    //========================Manual=============================
    modesMachine         := eMachineModes.Manual;
    expectedColor.Green  := FALSE;
    expectedColor.Red    := FALSE;
    expectedColor.Yellow := TRUE;

    actualColor := itfDut.SetMachineMode(modesMachine);

    AssertEquals
    (
        Expected  := expectedColor
        , Actual  := actualColor
        , Message := 'ColorOuput shall be Yellow'
    );

    //========================Fault=============================
    modesMachine         := eMachineModes.Fault;
    expectedColor.Green  := FALSE;
    expectedColor.Red    := TRUE;
    expectedColor.Yellow := FALSE;

     itfDut.SetMachineMode(modesMachine);
     actualColor := itfDut.GetColorsSignalLightMachineModes;
    AssertEquals
    (
        Expected  := expectedColor
        , Actual  := actualColor
        , Message := 'ColorOuput shall be Red'
    );

    state := 10;
END_IF

IF state = 10 THEN

    //========================Home=============================
    modesMachine := eMachineModes.Home;
    itfDut.SetMachineMode(modesMachine);

    IF eMachineModes.Home = modesMachine THEN
        timer(in := TRUE);
    END_IF

    expectedColor.Red    := FALSE;
    expectedColor.Yellow := FALSE;

    IF timer.ET >= 0 * blinkTime AND timer.ET < blinkTime THEN
        expectedColor.Green := TRUE;
        actualColor         := itfDut.SetMachineMode(modesMachine);

        AssertEquals
        (
            Expected  := expectedColor
            , Actual  := actualColor
            , Message := 'ColorOuput shall be GreenBlinking and True 1 '
        );

    ELSIF timer.ET > blinkTime + T#2MS AND timer.ET < 2 * blinkTime THEN
        expectedColor.Green := FALSE;
        actualColor         := itfDut.SetMachineMode(modesMachine);

        AssertEquals
        (
            Expected  := expectedColor
            , Actual  := actualColor
            , Message := 'ColorOuput shall be GreenBlinking and False 2'
        );

    ELSIF timer.ET > 2 * blinkTime + T#2MS AND timer.ET < 3 * blinkTime THEN
        expectedColor.Green := TRUE;
        actualColor         := itfDut.SetMachineMode(modesMachine);

        AssertEquals
        (
            Expected  := expectedColor
            , Actual  := actualColor
            , Message := 'ColorOuput shall be GreenBlinking and TRUE 3'
        );
    ELSIF timer.ET > 3 * blinkTime + T#2MS AND timer.ET < 4 * blinkTime THEN
        expectedColor.Green := False;
        actualColor         := itfDut.SetMachineMode(modesMachine);

        AssertEquals
        (
            Expected  := expectedColor
            , Actual  := actualColor
            , Message := 'ColorOuput shall be GreenBlinking and TRUE 4'
        );
    ELSIF timer.ET > 5 * blinkTime THEN

        //========================Idle, Check again if all out =============================
        modesMachine := eMachineModes.Idle;

        expectedColor.Green  := FALSE;
        expectedColor.Red    := FALSE;
        expectedColor.Yellow := FALSE;

        actualColor := itfDut.SetMachineMode(modesMachine);

        AssertEquals
        (
            Expected  := expectedColor
            , Actual  := actualColor
            , Message := 'ColorOuput shall be Off again'
        );

        {analysis -9}
        TEST_FINISHED();
    END_IF
END_IF
END_METHOD

PROPERTY StartCycleCount : ULINT
GET
StartCycleCount := THIS^._nfContext._startCycleCount;
END_GET
END_PROPERTY

END_FUNCTION_BLOCK

// ---- POUs/SignalLights MachineStatus/POUs/SignalLightsController.TcPOU
FUNCTION_BLOCK SignalLightsController EXTENDS TcoCore.TcoObject IMPLEMENTS ISignalLightsController
VAR
    blinker : Blinker;
    colorsStatus : ColorsSignalLightsStatus;
    colorsMode : ColorsSignalLightMachineModes;
END_VAR

METHOD FB_init : BOOL
VAR_INPUT
    bInitRetains : BOOL; // if TRUE, the retain variables are initialized (warm start / cold start)
    bInCopyCode  : BOOL; // if TRUE, the instance afterwards gets moved into the copy code (online change)
    ParentObject : ITcoObject;
END_VAR
END_METHOD

PROPERTY GetColorsSignalLightMachineModes :  ColorsSignalLightMachineModes
GET
GetColorsSignalLightMachineModes := colorsMode;
END_GET
END_PROPERTY

PROPERTY GetColorsSignalLightMachineStatus : ColorsSignalLightsStatus
GET
GetColorsSignalLightMachineStatus := colorsStatus;
END_GET
END_PROPERTY

(*~
    <docu>
        <summary>
            Restore all tasks of this instance into initial state.
        </summary>
    </docu>
~*)
METHOD Restore : ITcoRestorable
END_METHOD

METHOD PROTECTED ServiceMode
END_METHOD

METHOD SetBlinkTime
VAR_INPUT
    blinkOnTime  : TIME;
    blinkOffTime : TIME;
END_VAR
THIS^.blinker.SetOffTime(blinkOffTime);
THIS^.blinker.SetOnTime(blinkOnTime);
END_METHOD

METHOD SetMachineMode : ColorsSignalLightMachineModes
VAR_INPUT
    currentMachineMode : eMachineModes ;
END_VAR

IF eMachineModes.Home = currentMachineMode THEN
    blinker.ExecuteTimer();
END_IF

CASE currentMachineMode OF
    eMachineModes.Fault:
        colorsMode.Red    := TRUE;
        colorsMode.Green  := FALSE;
        colorsMode.Yellow := FALSE;

    eMachineModes.Idle:

        colorsMode.Red    := FALSE;
        colorsMode.Green  := FALSE;
        colorsMode.Yellow := FALSE;

    eMachineModes.Automat:
        colorsMode.Red    := FALSE;
        colorsMode.Green  := TRUE;
        colorsMode.Yellow := FALSE;

    eMachineModes.Step:
        colorsMode.Red    := FALSE;
        colorsMode.Green  := TRUE;
        colorsMode.Yellow := TRUE;

    eMachineModes.Home:
        colorsMode.Red    := FALSE;
        colorsMode.Yellow := FALSE;
        colorsMode.Green  := blinker.IsOn;

    eMachineModes.Manual:
        colorsMode.Red    := FALSE;
        colorsMode.Yellow := TRUE;
        colorsMode.Green  := FALSE;
ELSE
    ;
END_CASE

 SetMachineMode := colorsMode ;
END_METHOD

METHOD SetMachineStatusOff : ColorsSignalLightsStatus
VAR_INPUT
    currentMachineStatus : eMachineStatus;
END_VAR
CASE currentMachineStatus OF
    eMachineStatus.Blue:
        colorsStatus.Blue := FALSE;
    eMachineStatus.Turquise:
        colorsStatus.Turquise := FALSE;
    eMachineStatus.Violet:
        colorsStatus.Violet := FALSE;
    eMachineStatus.White:
        colorsStatus.White := FALSE;
    eMachineStatus.All:
        colorsStatus.Blue     := FALSE;
        colorsStatus.Turquise := FALSE;
        colorsStatus.White    := FALSE;
        colorsStatus.Violet   := FALSE;
END_CASE

SetMachineStatusOff := colorsStatus;
END_METHOD

METHOD SetMachineStatusOn : ColorsSignalLightsStatus
VAR_INPUT
    currentMachineStatus : eMachineStatus;
END_VAR
CASE currentMachineStatus OF
    eMachineStatus.Blue:
        colorsStatus.Blue := TRUE;
    eMachineStatus.Turquise:
        colorsStatus.Turquise := TRUE;
    eMachineStatus.Violet:
        colorsStatus.Violet := TRUE;
    eMachineStatus.White:
        colorsStatus.White := TRUE;
    eMachineStatus.All:
        colorsStatus.Blue     := TRUE;
        colorsStatus.Turquise := TRUE;
        colorsStatus.White    := TRUE;
        colorsStatus.Violet   := TRUE;
END_CASE

SetMachineStatusOn := colorsStatus;
END_METHOD

END_FUNCTION_BLOCK

// ---- POUs/Utilities/Blinker.TcPOU
FUNCTION_BLOCK Blinker
VAR
    _offTime : TIME := T#1000MS;
    _onTime  : TIME := T#1000MS;
    onTimer : TON;
    offTimer : TON;
    blinkOutput : BOOL;
    state : INT ;
END_VAR

METHOD ExecuteTimer : BOOL
VAR_INPUT
END_VAR
IF state = 0 THEN
    onTimer(in := FALSE);
    offTimer(in := FALSE);

    state := 10;
END_IF

IF state = 10 THEN
    onTimer(in := TRUE, pt := _onTime);
    blinkOutput := TRUE;

    IF onTimer.Q THEN
        state := 20;

        RETURN;
    END_IF
END_IF

IF state = 20 THEN
    offTimer(in := TRUE, pt := _offTime);
    blinkOutput := FALSE;

    IF offTimer.Q THEN
        state := 0;
    END_IF
END_IF
END_METHOD

PROPERTY IsOn : BOOL
GET
IsOn := blinkOutput;
END_GET
END_PROPERTY

METHOD SetOffTime
VAR_INPUT
    offTime : TIME;
END_VAR
_offTime := offTime;
END_METHOD

METHOD SetOnTime
VAR_INPUT
    onTime: TIME;
END_VAR
_onTime := onTime;
END_METHOD

END_FUNCTION_BLOCK

// ---- Test/BlinkerTest/Blinker_Test.TcPOU
FUNCTION_BLOCK Blinker_Test EXTENDS TcUnit.FB_TestSuite

ExecuteBlinker_ExpectBlinkingWithSetTime();

METHOD PRIVATE ExecuteBlinker_ExpectBlinkingWithSetTime
VAR_INST
    dut : Blinker;
    timeOn : TIME ;
    timeOff : TIME;
    duration : TIME;
    ReferenceTimerOn : TON;
    ReferenceTimerOff : TON;

    state : INT;
    expectedResult : BOOL;
    actualResult : BOOL;
END_VAR
TEST('ExecuteBlinker_ExpectBlinkingWithSetTime');
timeOn  := T#2MS;
timeOff := T#5MS;
dut.SetOffTime(timeOff);
dut.SetOnTime(timeOn);
ReferenceTimerOn();
ReferenceTimerOff();
dut.ExecuteTimer();

IF state = 0 THEN
    ReferenceTimerOn(in := TRUE, pt := 2 * timeOn);

    AssertTrue(dut.IsOn, 'Shall be True');
    state := 10;
END_IF

IF state = 10 THEN
    IF ReferenceTimerOn.ET = timeOn THEN
        AssertTrue(dut.IsOn, 'Shall be True State 10');
        state := 20;
        ReferenceTimerOn(in := FALSE);
        ReferenceTimerOff(in := TRUE, pt := 2 * timeOff);
        RETURN;
    END_IF
END_IF

IF state = 20 THEN
    AssertFalse(dut.IsOn, 'Shall be False');

    IF ReferenceTimerOff.ET = timeOff THEN
        AssertFalse(dut.IsOn, 'Shall still be Falsem, State 20');
        state := 30;
        ReferenceTimerOff(in := FALSE);
        ReferenceTimerOn(in := TRUE);
        RETURN;
    END_IF
END_IF

IF state = 30 THEN
    IF ReferenceTimerOn.ET = timeOn THEN
        AssertTrue(dut.IsOn, 'Shall be True State 20');
        state := 40;
        ReferenceTimerOn(in := FALSE);
        RETURN;
    END_IF
END_IF

IF state = 40 THEN
    {analysis -9}
    TEST_FINISHED();

END_IF
END_METHOD

END_FUNCTION_BLOCK

// ---- Test/CounterAllgemeinTests/Counter_Test.TcPOU
FUNCTION_BLOCK INTERNAL Counter_Test EXTENDS TcUnit.FB_TestSuite IMPLEMENTS TcoCore.ITcoContext
VAR
    //Context for TcOpen
    _nfContext : TcoCore.TcoContextNfCompatibility;
END_VAR

SetInitalValueExpectThisValueAsResult();
InitalFbCountUpToLimitExpectCorrespondingValuesAndProp();
CountDownToZeroExpectCorrespondingPropAndValue();
CountUpDownBy10ExpectCorrespondingValue();
ResetExpectNull();

PROPERTY Context : TcoCore.ITcoContext
GET
Context := This^._nfContext;
END_GET
END_PROPERTY

METHOD PRIVATE CountDownToZeroExpectCorrespondingPropAndValue
VAR_INST
    dut    : Counter(THIS^, countStep := 1, countInitValue := 3, countLimit := 7);
    itfDut : ICounter;

    expected : StatusCounter;
    actual   : StatusCounter;

    valueEx :UDINT;
    valueAc : UDINT;

    reached : BOOL;

END_VAR
TEST('CountDownToZeroExpectCorrespondingPropAndValue');

//Arrange
IF itfDut = 0 THEN
    itfDut := dut;
END_IF


itfDut.CountDown();

valueEx := 2;
valueAc := itfDut.CountValue;

AssertEquals_UDINT(valueEx, valueAc, 'Value muss 2 sein ');


itfDut.CountDown();

valueEx := 1;
valueAc := itfDut.CountValue;

AssertEquals_UDINT(valueEx, valueAc, 'Value muss 1 sein ');

itfDut.CountDown();

valueEx := 0;
valueAc := itfDut.CountValue;

AssertEquals_UDINT(valueEx, valueAc, 'Value muss 1 sein ');
reached := itfDut.CountLimitReached;

AssertTrue(itfDut.CountZeroReached, 'CountZeroReached muss True sein');


{analysis -9}
TEST_FINISHED();
END_METHOD

METHOD PRIVATE CountUpDownBy10ExpectCorrespondingValue
VAR_INST
    dut    : Counter(THIS^, countStep := 10, countInitValue := 0, countLimit := 15);
    itfDut : ICounter;

    expected : StatusCounter;
    actual   : StatusCounter;

    valueEx :UDINT;
    valueAc : UDINT;

    reached : BOOL;

END_VAR
TEST('CountUpDownBy10ExpectCorrespondingValue');

//Arrange
IF itfDut = 0 THEN
    itfDut := dut;
END_IF

valueEx := 0;
valueAc := itfDut.CountValue;

AssertEquals_UDINT(valueEx, valueAc, 'Value muss 0 sein ');

///////////////////////////
itfDut.CountUp();

valueEx := 10;
valueAc := itfDut.CountValue;
AssertEquals_UDINT(valueEx, valueAc, 'Value muss 10 sein ');
AssertFalse(itfDut.CountLimitReached, 'countLimitReached muss False sein');

itfDut.CountUp();

valueEx := 20;
valueAc := itfDut.CountValue;

AssertEquals_UDINT(valueEx, valueAc, 'Value muss 20 sein ');

AssertTrue(itfDut.CountLimitReached, 'countLimitReached muss True sein');
AssertFalse(itfDut.CountZeroReached, 'CountZeroReached muss False sein');

/////////////////////////////
itfDut.CountDown();
itfDut.CountDown();

valueEx := 0;
valueAc := itfDut.CountValue;

AssertEquals_UDINT(valueEx, valueAc, 'Value muss 0 sein ');

AssertFalse(itfDut.CountLimitReached, 'countLimitReached muss False sein');
AssertTrue(itfDut.CountZeroReached, 'CountZeroReached muss TRUE sein');

{analysis -9}
TEST_FINISHED();
END_METHOD

PROPERTY EndCycleCount : ULINT
GET
EndCycleCount := THIS^._nfContext._endCycleCount;
END_GET
END_PROPERTY

PROPERTY Environment : TcoCore.ITcoContextEnvironment
GET
Environment := THIS^._nfContext._settings;
END_GET
END_PROPERTY

PROPERTY Identity : ULINT
GET
Identity := THIS^._nfContext._Identity;
END_GET
END_PROPERTY

METHOD PRIVATE InitalFbCountUpToLimitExpectCorrespondingValuesAndProp
VAR_INST
    dut    : Counter(THIS^, countStep := 1, countInitValue := 5, countLimit := 7);
    itfDut : ICounter;

    expected : StatusCounter;
    actual   : StatusCounter;

    valueEx :UDINT;
    valueAc : UDINT;

    reached : BOOL;

END_VAR
TEST('InitalFbCountUpToLimitExpectCorrespondingValuesAndProp');

//Arrange
IF itfDut = 0 THEN
    itfDut := dut;
END_IF


itfDut.CountUp();

valueEx := 6;
valueAc := itfDut.CountValue;

AssertEquals_UDINT(valueEx, valueAc, 'Value muss 6 sein ');

itfDut.CountUp();

valueEx := 7;
valueAc := itfDut.CountValue;

AssertEquals_UDINT(valueEx, valueAc, 'Value muss 7 sein ');

reached := itfDut.CountLimitReached;

AssertTrue(reached, 'countLimitReached muss True sein');
AssertFalse(itfDut.CountZeroReached, 'CountZeroReached muss False sein');

{analysis -9}
TEST_FINISHED();
END_METHOD

PROPERTY Logger : TcoCore.ITcoLogger
GET
Logger := THIS^._nfContext._logger;
END_GET
END_PROPERTY

PROPERTY RealTimeClock : TcoCore.ITcoRtc
GET
RealTimeClock := THIS^._nfContext._rtc;
END_GET
END_PROPERTY

METHOD PRIVATE ResetExpectNull
VAR_INST
    dut    : Counter(THIS^, countStep := 10, countInitValue := 0, countLimit := 15);
    itfDut : ICounter;

    expected : StatusCounter;
    actual   : StatusCounter;

    valueEx :UDINT;
    valueAc : UDINT;

    reached : BOOL;

END_VAR
TEST('ResetExpectNull');

//Arrange
IF itfDut = 0 THEN
    itfDut := dut;
END_IF

valueEx := 0;
valueAc := itfDut.CountValue;

AssertEquals_UDINT(valueEx, valueAc, 'Value muss 0 sein ');

///////////////////////////
itfDut.CountUp();

valueEx := 10;
valueAc := itfDut.CountValue;
AssertEquals_UDINT(valueEx, valueAc, 'Value muss 10 sein ');
AssertFalse(itfDut.CountLimitReached, 'countLimitReached muss False sein');

itfDut.CountUp();

valueEx := 20;
valueAc := itfDut.CountValue;

AssertEquals_UDINT(valueEx, valueAc, 'Value muss 20 sein ');

itfDut.ResetCount();

valueEx :=0;
valueAc := itfDut.CountValue;
AssertTrue(itfDut.CountZeroReached, 'nach Reset muss Zero sein');
AssertEquals_UDINT(valueEx, valueAc, 'Value muss 0 sein ');

{analysis -9}
TEST_FINISHED();
END_METHOD

METHOD PRIVATE SetInitalValueExpectThisValueAsResult
VAR_INST
    dut    : Counter(THIS^, countStep := 1, countInitValue := 5, countLimit := 10);
    itfDut : ICounter;
 status : StatusCounter;

END_VAR
TEST('SetInitalValueExpectThisValueAsResult');


//Arrange
IF itfDut = 0 THEN
    itfDut := dut;
END_IF

//Aact

// Assert

AssertEquals_UDINT(5, itfdut.CountValue, 'Value should be 5');

{analysis -9}
TEST_FINISHED();
END_METHOD

PROPERTY StartCycleCount : ULINT
GET
StartCycleCount := THIS^._nfContext._startCycleCount;
END_GET
END_PROPERTY

END_FUNCTION_BLOCK

// ---- POUs/Cylinders/Base/TcoDoubleCylinderBase.TcPOU
FUNCTION_BLOCK ABSTRACT TcoDoubleCylinderBase EXTENDS TcoCore.TcoComponent IMPLEMENTS ITcoCylinder
VAR_IN_OUT
    (*~
        <docu>
            <summary>
                Home position sensor 1.
            </summary>
        </docu>
    ~*)
    {attribute addProperty Name "<#Home position sensor#> - 1"}
    inoAtHomePos1 : BOOL;
    (*~
        <docu>
            <summary>
                Home position sensor 2.
            </summary>
        </docu>
    ~*)
    {attribute addProperty Name "<#Home position sensor#> - 2"}
    inoAtHomePos2 : BOOL;
    (*~
        <docu>
            <summary>
                Working position sensor 1.
            </summary>
        </docu>
    ~*)
    {attribute addProperty Name "<#Work position sensor#> - 1"}
    inoAtWorkPos1 : BOOL;
    (*~
        <docu>
            <summary>
                Working position sensor 1.
            </summary>
        </docu>
    ~*)
    {attribute addProperty Name "<#Work position sensor#> - 2"}
    inoAtWorkPos2 : BOOL;
END_VAR
VAR_IN_OUT
    (*~
        <docu>
            <summary>
                Move to working home position signal.
            </summary>
        </docu>
    ~*)
    {attribute addProperty Name "<#Move to home position actuator#>"}
    inoToHomePos : BOOL;
    (*~
        <docu>
            <summary>
                Move to working posistion signal.
            </summary>
        </docu>
    ~*)
    {attribute addProperty Name "<#Move to work position actuator#>"}
    inoToWorkPos : BOOL;
END_VAR
VAR
    (*~
        <docu>
            <summary>
                Home position sensor.
            </summary>
        </docu>
    ~*)
    {attribute addProperty Name "<#Home position sensor#>"}
    _atHomePos : BOOL;
    (*~
        <docu>
            <summary>
                Working position sensor.
            </summary>
        </docu>
    ~*)
    {attribute addProperty Name "<#Work position sensor#>"}
    _atWorkPos : BOOL;
    (*~
        <docu>
            <summary>
                Move to working home position signal.
            </summary>
        </docu>
    ~*)
    {attribute addProperty Name "<#Move to home position actuator#>"}
    _toHomePos : BOOL;
    (*~
        <docu>
            <summary>
                Move to working posistion signal.
            </summary>
        </docu>
    ~*)
    {attribute addProperty Name "<#Move to work position actuator#>"}
    _toWorkPos : BOOL;
END_VAR

VAR
    {attribute addProperty Name "<#Home sensor signal 1#>"}
    _atHomePos1SignalInfo : TcoCore.TcoSignalInfo;
    {attribute addProperty Name "<#Home sensor signal 2#>"}
    _atHomePos2SignalInfo : TcoCore.TcoSignalInfo;
    {attribute addProperty Name "<#Work sensor signal 1#>"}
    _atWorkPos1SignalInfo : TcoCore.TcoSignalInfo;
    {attribute addProperty Name "<#Work sensor signal 2#>"}
    _atWorkPos2SignalInfo : TcoCore.TcoSignalInfo;
    {attribute addProperty Name "<#Move to home position signal#>"}
    _toHomePosSignalInfo : TcoCore.TcoSignalInfo;
    {attribute addProperty Name "<#Move to work position signal#>"}
    _toWorkPosSignalInfo : TcoCore.TcoSignalInfo;
END_VAR

IF (__ISVALIDREF(inoAtHomePos1) AND __ISVALIDREF(inoAtHomePos2)) THEN
    _atHomePos := inoAtHomePos1 AND inoAtHomePos2;
    _atHomePos1SignalInfo.GetSignalInfo(SIZEOF(inoAtHomePos1), ADR(inoAtHomePos1));
    _atHomePos2SignalInfo.GetSignalInfo(SIZEOF(inoAtHomePos2), ADR(inoAtHomePos2));
END_IF;

IF (__ISVALIDREF(inoAtWorkPos1) AND __ISVALIDREF(inoAtWorkPos2)) THEN
    _atWorkPos := inoAtWorkPos1 AND inoAtWorkPos2;
    _atWorkPos1SignalInfo.GetSignalInfo(SIZEOF(inoAtWorkPos1), ADR(inoAtWorkPos1));
    _atWorkPos2SignalInfo.GetSignalInfo(SIZEOF(inoAtWorkPos2), ADR(inoAtWorkPos2));
END_IF;

IF (__ISVALIDREF(inoToHomePos)) THEN
    inoToHomePos := _toHomePos;
    _toHomePosSignalInfo.GetSignalInfo(SIZEOF(inoToHomePos), ADR(inoToHomePos));
END_IF;

IF (__ISVALIDREF(inoToWorkPos)) THEN
    inoToWorkPos := _toWorkPos;
    _toWorkPosSignalInfo.GetSignalInfo(SIZEOF(inoToWorkPos), ADR(inoToWorkPos));
END_IF;

(*~
    <docu>
        <summary>
            Gets whether the piston is in home position.
        </summary>
    </docu>
~*)
PROPERTY AtHome : bool
GET
AtHome := THIS^._atHomePos;
END_GET
END_PROPERTY

(*~
    <docu>
        <summary>
            Gets whether the piston is in work position.
        </summary>
    </docu>
~*)
PROPERTY AtWork : bool
GET
AtWork := _atWorkPos;
END_GET
END_PROPERTY

METHOD FB_init : BOOL
VAR_INPUT
    bInitRetains : BOOL; // if TRUE, the retain variables are initialized (warm start / cold start)
    bInCopyCode  : BOOL; // if TRUE, the instance afterwards gets moved into the copy code (online change)
    ParentObject : ITcoObject;
END_VAR
END_METHOD

(*~
    <docu>
        <summary>
            Gets the `MoveHomeTask` task that controls the moving of the cyclinder in home position.
            <remarks>
                <note type="important">
                    This is an abstract method and must be implemented in derived class.
                </note>
            </remarks>
        </summary>
    </docu>
~*)
PROPERTY PUBLIC ABSTRACT MoveHomeTask : TcoCore.ITcoTask
GET
END_GET
END_PROPERTY

(*~
    <docu>
        <summary>
            Starts movement into home position.
        </summary>
    </docu>
~*)
METHOD MoveToHome : TcoCore.ITcoTaskStatus
IF (MoveHomeTask <> 0) THEN
    MoveToHome := MoveHomeTask.Invoke();
END_IF;
END_METHOD

(*~
    <docu>
        <summary>
            Starts movement into work position.
        </summary>
    </docu>
~*)
METHOD MoveToWork : TcoCore.ITcoTaskStatus
IF (MoveWorkTask <> 0) THEN
    MoveToWork := MoveWorkTask.Invoke();
END_IF;
END_METHOD

(*~
    <docu>
        <summary>
            Gets the `MoveWorkTask` task that controls the moving of the cyclinder into work position.
            <remarks>
                <note type="important">
                    This is an abstract method and must be implemented in derived class.
                </note>
            </remarks>
        </summary>
    </docu>
~*)
PROPERTY PUBLIC ABSTRACT MoveWorkTask : TcoCore.ITcoTask
GET
END_GET
END_PROPERTY

(*~
    <docu>
        <summary>
            Restore all tasks of this instance into initial state.
        </summary>
    </docu>
~*)
METHOD Restore : ITcoRestorable
IF (MoveHomeTask <> 0) THEN
    MoveHomeTask.Restore();
END_IF;

IF (MoveWorkTask <> 0) THEN
    MoveWorkTask.Restore();
END_IF;

IF (StopTask <> 0) THEN
    StopTask.Restore();
END_IF;
END_METHOD

METHOD PROTECTED ServiceMode
END_METHOD

(*~
    <docu>
        <summary>
            Stops cyclinder movement.
             <remarks>
                <note type="important">
                    This method switched off the signals for the movement of the piston in both direction.
                    However depending on the pnemumatics configuration the movement may contintue if designed in that way.
                    THIS IS NOT A SAFETY FUCTION!
                </note>
            </remarks>
        </summary>
    </docu>
~*)
METHOD Stop : TcoCore.ITcoTaskStatus
IF (StopTask <> 0) THEN
    Stop := StopTask.Invoke();
END_IF;
END_METHOD

(*~
    <docu>
        <summary>
            Gets the `StopTask` task that controls the stopping cyclinder movement.
            <remarks>
                <note type="important">
                    This is an abstract method and must be implemented in derived class.
                </note>
            </remarks>
        </summary>
    </docu>
~*)
PROPERTY PUBLIC ABSTRACT StopTask : TcoCore.ITcoTask
GET
END_GET
END_PROPERTY

END_FUNCTION_BLOCK

// ---- POUs/Cylinders/ExampleCylinder/ExampleCylinder.TcPOU
(*~
        <docu>
            <summary>
                This is an example implementation of `ExampleCyclinder` component.
            </summary>
        </docu>
~*)
FUNCTION_BLOCK ExampleCylinder EXTENDS TcoCore.TcoComponent
VAR_IN_OUT
    (*~
        <docu>
            <summary>
                Home position sensor.
            </summary>
        </docu>
    ~*)
    {attribute addProperty Name "<#Home position sensor#>"}
    inoAtHomePos : BOOL;
    (*~
        <docu>
            <summary>
                Working position sensor.
            </summary>
        </docu>
    ~*)
    {attribute addProperty Name "<#Work position sensor#>"}
    inoAtWorkPos : BOOL;
    (*~
        <docu>
            <summary>
                Move to working home position signal.
            </summary>
        </docu>
    ~*)
    {attribute addProperty Name "<#Move to home position actuator#>"}
    inoToHomePos : BOOL;
    (*~
        <docu>
            <summary>
                Move to working posistion signal.
            </summary>
        </docu>
    ~*)
    {attribute addProperty Name "<#Move to work position actuator#>"}
    inoToWorkPos : BOOL;
END_VAR
VAR
    (*~
        <docu>
            <summary>
                Home position sensor.
            </summary>
        </docu>
    ~*)
    {attribute addProperty Name "<#Home position sensor#>"}
    _atHomePos : BOOL;
    (*~
        <docu>
            <summary>
                Working position sensor.
            </summary>
        </docu>
    ~*)
    {attribute addProperty Name "<#Work position sensor#>"}
    _atWorkPos : BOOL;
    (*~
        <docu>
            <summary>
                Move to working home position signal.
            </summary>
        </docu>
    ~*)
    {attribute addProperty Name "<#Move to home position actuator#>"}
    _toHomePos : BOOL;
    (*~
        <docu>
            <summary>
                Move to working posistion signal.
            </summary>
        </docu>
    ~*)
    {attribute addProperty Name "<#Move to work position actuator#>"}
    _toWorkPos : BOOL;
END_VAR

VAR
    _atHomePosSignalInfo : TcoCore.TcoSignalInfo;
    _atWorkPosSignalInfo : TcoCore.TcoSignalInfo;
    _toHomePosSignalInfo : TcoCore.TcoSignalInfo;
    _toWorkPosSignalInfo : TcoCore.TcoSignalInfo;
END_VAR

VAR
    {attribute addProperty Name "<#Move Home#>"}
    _moveHomeDefault : ExampleCylinderMoveTask(THIS^);
    {attribute addProperty Name "<#Move to Work#>"}
    _moveWorkDefault : ExampleCylinderMoveTask(THIS^);
    {attribute addProperty Name "<#Stop#>"}
    _stopDefault : TcoCore.TcoTask(THIS^);
END_VAR
VAR
    _config : TcoCylinderConfig;
    _status : TcoCylinderStatus;
END_VAR

// Updates I/O
UpdateIO();

// Disables mutualy exclusive actions
_moveWorkDefault.Enabled := NOT _moveHomeDefault.Busy;

_moveHomeDefault
(
    PositionSensor           := _atHomePos
    , MoveToPositionSignal   := _toHomePos
    , InverseSignal          := _toWorkPos
    , MaxTimeToReachPosition := _config.TimeToReachHomePosition
    , PositionName           := '<#Home#>'
);

// Disables mutualy exclusive actions
_moveHomeDefault.Enabled := NOT _moveWorkDefault.Busy;

_moveWorkDefault
(
    PositionSensor           := _atWorkPos
    , MoveToPositionSignal   := _toWorkPos
    , InverseSignal          := _toHomePos
    , MaxTimeToReachPosition := _config.TimeToReachWorkPosition
    , PositionName           := '<#Work#>'
);

IF (_stopDefault.Execute()) THEN
    _toHomePos := FALSE;
    _toWorkPos := FALSE;
    _moveHomeDefault.Abort();
    _moveWorkDefault.Abort();
    _stopDefault.Abort();
    _moveHomeDefault.Restore();
    _moveWorkDefault.Restore();
    _stopDefault.Restore();
    _stopDefault.DoneWhen(TRUE);
END_IF

// For further discussion about Status
IF (_moveHomeDefault.Busy) THEN
    _status.ActionDescription := 'Moving to home position';
ELSIF (_moveWorkDefault.Busy) THEN
    _status.ActionDescription := 'Moving to work position';
ELSIF (_stopDefault.Busy) THEN
    _status.ActionDescription := 'Stopping pressure';
ELSE
    _status.ActionDescription := 'Idle';
END_IF

UpdateIO();

(*~
    <docu>
        <summary>
            Gets whether the piston is in home position.
        </summary>
    </docu>
~*)
PROPERTY AtHome : bool
GET
AtHome := THIS^._atHomePos;
END_GET
END_PROPERTY

(*~
    <docu>
        <summary>
            Gets whether the piston is in work position.
        </summary>
    </docu>
~*)
PROPERTY AtWork : bool
GET
AtWork := _atWorkPos;
END_GET
END_PROPERTY

(*~
    <docu>
        <summary>
            Gets the configuration of the cylinder.
        </summary>
    </docu>
~*)
PROPERTY Config : REFERENCE TO TcoCylinderConfig
GET
Config REF= config;
END_GET
END_PROPERTY

(*~
    <docu>
        <summary>
            Gets the `MoveHomeTask` task that controls the moving of the cyclinder in home position.
        </summary>
    </docu>
~*)
PROPERTY MoveHomeTask : TcoCore.ITcoTask
GET
MoveHomeTask := _moveHomeDefault;
END_GET
END_PROPERTY

(*~
    <docu>
        <summary>
            Starts movement into home position.
        </summary>
    </docu>
~*)
METHOD MoveToHome : TcoCore.ITcoTaskStatus
IF (MoveHomeTask <> 0) THEN
    MoveToHome := MoveHomeTask.Invoke();
END_IF;
END_METHOD

(*~
    <docu>
        <summary>
            Starts movement into work position.
        </summary>
    </docu>
~*)
METHOD MoveToWork : TcoCore.ITcoTaskStatus
IF (MoveWorkTask <> 0) THEN
    MoveToWork := MoveWorkTask.Invoke();
END_IF;
END_METHOD

(*~
    <docu>
        <summary>
            Gets the `MoveWorkTask` task that controls the moving of the cyclinder into work position.
        </summary>
    </docu>
~*)
PROPERTY MoveWorkTask : TcoCore.ITcoTask
GET
MoveWorkTask := _moveWorkDefault;
END_GET
END_PROPERTY

(*~
    <docu>
        <summary>
            Restores this instance to the Ready state. Can be called explicitly or from within one of the restore mechanisms.
        </summary>
    </docu>
~*)
METHOD Restore : ITcoRestorable
IF (MoveHomeTask <> 0) THEN
    MoveHomeTask.Restore();
END_IF;

IF (MoveWorkTask <> 0) THEN
    MoveWorkTask.Restore();
END_IF;

IF (StopTask <> 0) THEN
    StopTask.Restore();
END_IF;
END_METHOD

(*~
    <docu>
        <summary>
            Custom service (manual, maintenance) logic.
            This method must be implemented in derived class.
        </summary>
    </docu>
~*)
METHOD PROTECTED ServiceMode
END_METHOD

PROPERTY Status : REFERENCE TO TcoCylinderStatus
GET
Status REF= _status;
END_GET
END_PROPERTY

(*~
    <docu>
        <summary>
            Stops cyclinder movement.
             <remarks>
                <note type="important">
                    This method switched off the signals for the movement of the piston in both direction.
                    However depending on the pnemumatics configuration the movement may contintue if designed in that way.
                    THIS IS NOT A SAFETY FUCTION!
                </note>
            </remarks>
        </summary>
    </docu>
~*)
METHOD Stop : TcoCore.ITcoTaskStatus
IF (StopTask <> 0) THEN
    Stop := StopTask.Invoke();
END_IF;
END_METHOD

(*~
    <docu>
        <summary>
            Gets the `StopTask` task that controls the stopping of the cyclinder.
        </summary>
    </docu>
~*)
PROPERTY StopTask : TcoCore.ITcoTask
GET
StopTask := _stopDefault;
END_GET
END_PROPERTY

METHOD PRIVATE UpdateIO
IF (__ISVALIDREF(inoAtHomePos)) THEN
    _atHomePos := inoAtHomePos;
    _atHomePosSignalInfo.GetSignalInfo(SIZEOF(inoAtHomePos), ADR(inoAtHomePos));
END_IF;

IF (__ISVALIDREF(inoAtWorkPos)) THEN
    _atWorkPos := inoAtWorkPos;
    _atWorkPosSignalInfo.GetSignalInfo(SIZEOF(inoAtWorkPos), ADR(inoAtWorkPos));
END_IF;

IF (__ISVALIDREF(inoToHomePos)) THEN
    inoToHomePos := _toHomePos;
    _toHomePosSignalInfo.GetSignalInfo(SIZEOF(inoToHomePos), ADR(inoToHomePos));
END_IF;

IF (__ISVALIDREF(inoToWorkPos)) THEN
    inoToWorkPos := _toWorkPos;
    _toWorkPosSignalInfo.GetSignalInfo(SIZEOF(inoToWorkPos), ADR(inoToWorkPos));
END_IF;
END_METHOD

END_FUNCTION_BLOCK

// ---- POUs/Cylinders/ExampleCylinder/ExampleCylinderMoveTask.TcPOU
FUNCTION_BLOCK ExampleCylinderMoveTask EXTENDS TcoCore.TcoTask
VAR_INPUT
    PositionSensor         : BOOL;
    MaxTimeToReachPosition : TIME := T#10S;
    PositionName           : STRING(25);
END_VAR
VAR_IN_OUT
    MoveToPositionSignal : BOOL;
    InverseSignal        : BOOL;
END_VAR

VAR
    _stringBuilder : TcoCore.StringBuilder;
END_VAR

IF (THIS^.Execute()) THEN
    IF (THIS^.ElapsedTime > MaxTimeToReachPosition) THEN
        THIS^.Messenger
            .Warning(_stringBuilder.Clear().Append(PositionName).Append(' sensor not reached yet.').ToString());
    END_IF;

    InverseSignal        := FALSE;
    MoveToPositionSignal := TRUE;
    THIS^.DoneWhen(PositionSensor);
END_IF

METHOD PUBLIC FB_init : BOOL
VAR_INPUT
    bInitRetains : BOOL; // if TRUE, the retain variables are initialized (warm start / cold start)
    bInCopyCode  : BOOL; // if TRUE, the instance afterwards gets moved into the copy code (online change)
    ParentObject : ITcoObject;
END_VAR
END_METHOD

(*~
    <docu>
        <summary>
            Executes when task is aborted.
        </summary>
    </docu>
~*)
METHOD PROTECTED OnAbort
MoveToPositionSignal := FALSE;
END_METHOD

METHOD PROTECTED OnError
END_METHOD

END_FUNCTION_BLOCK

// ---- POUs/Cylinders/TcoDoubleCylinder.TcPOU
{attribute addProperty _moveHomeDefaultName "<#MOVE HOME#>"}
{attribute addProperty _moveWorkDefaultName "<#MOVE TO WORK#>"}
{attribute addProperty _stopDefaultName "<#STOP#>"}
FUNCTION_BLOCK TcoDoubleCylinder EXTENDS TcoDoubleCylinderBase
VAR
    {attribute addProperty Name "|[[1]Attribute_moveHomeDefaultName]|"}
    _moveHomeDefault : TcoCylinderMoveTask(THIS^);
    {attribute addProperty Name "|[[1]Attribute_moveWorkDefaultName]|"}
    _moveWorkDefault : TcoCylinderMoveTask(THIS^);
    {attribute addProperty Name "|[[1]Attribute_stopDefaultName]|"}
    _stopDefault : TcoCore.TcoTask(THIS^);
    increment    : INT;

END_VAR
VAR
    _config      : TcoCylinderConfig;
    _status      : TcoCylinderStatus;
    _refillTimer : TON;
END_VAR

SUPER^
(
    inoAtHomePos1   := inoAtHomePos1
    , inoAtHomePos2 := inoAtHomePos2
    , inoAtWorkPos1 := inoAtWorkPos1
    , inoAtWorkPos2 := inoAtWorkPos2
    , inoToHomePos  := inoToHomePos
    , inoToWorkPos  := inoToWorkPos
);

IF (_atHomePos AND _atWorkPos) THEN
    Messenger.Error('<#Home and work position sensors are both active. Check the position of sensors!#>');
END_IF;

// Disables mutualy exclusive actions
_moveWorkDefault.Enabled := TRUE; // NOT _moveHomeDefault.Busy;

_moveHomeDefault
(
    PositionSensor           := _atHomePos AND NOT _atWorkPos
    , MoveToPositionSignal   := _toHomePos
    , InverseSignal          := _toWorkPos
    , TimeToRefill           := _config.TimeToRefill
    , MaxTimeToReachPosition := _config.TimeToReachHomePosition
    , PositionName           := '<#Home#>'
);

IF _moveHomeDefault.Execute() THEN
    _moveWorkDefault.Restore();
END_IF

// Disables mutualy exclusive actions
_moveHomeDefault.Enabled := true; // NOT _moveWorkDefault.Busy;

_moveWorkDefault
(
    PositionSensor           := _atWorkPos AND NOT _atHomePos
    , MoveToPositionSignal   := _toWorkPos
    , InverseSignal          := _toHomePos
    , TimeToRefill           := _config.TimeToRefill
    , MaxTimeToReachPosition := _config.TimeToReachWorkPosition
    , PositionName           := '<#Work#>'
);

IF _moveWorkDefault.Execute() THEN
    _moveHomeDefault.Restore();
END_IF

IF (_stopDefault.Execute()) THEN
    _toHomePos := FALSE;
    _toWorkPos := FALSE;
    _moveHomeDefault.Abort();
    _moveWorkDefault.Abort();
    _stopDefault.Abort();
    _moveHomeDefault.Restore();
    _moveWorkDefault.Restore();
    _stopDefault.Restore();
    _stopDefault.DoneWhen(TRUE);
END_IF

// For further discussion about Status
IF (_moveHomeDefault.Busy) THEN
    _status.ActionDescription := 'Moving to home position';
ELSIF (_moveWorkDefault.Busy) THEN
    _status.ActionDescription := 'Moving to work position';
ELSIF (_stopDefault.Busy) THEN
    _status.ActionDescription := 'Stopping pressure';
ELSE
    _status.ActionDescription := 'Idle';
END_IF

SUPER^
(
    inoAtHomePos1   := inoAtHomePos1
    , inoAtHomePos2 := inoAtHomePos2
    , inoAtWorkPos1 := inoAtWorkPos1
    , inoAtWorkPos2 := inoAtWorkPos2
    , inoToHomePos  := inoToHomePos
    , inoToWorkPos  := inoToWorkPos
);

(*~
    <docu>
        <summary>
            Aborts the movement to home position when the condition is 'true'.
        </summary>
        <remarks>
                <note type="warning">
                    The call of this method will be effective only when called AFTER the initialization of the instance of given TcoCylinder.
                </note>
        </remarks>
    </docu>
~*)
METHOD AbortMoveHome : BOOL
VAR_IN_OUT
    (*~
    <docu>
        <summary>
            Condition to abort the movement of the cylinder.
        </summary>
    </docu>
    ~*)
    inoDisableCondition : BOOL;
END_VAR
VAR
    _signalInfo : TcoSignalInfo;
END_VAR
IF (_toHomePos OR _moveHomeDefault.Busy) AND inoDisableCondition THEN
    _signalInfo.GetSignalInfo(SIZEOF(inoDisableCondition), ADR(inoDisableCondition));
    Messenger.Build().Append('<#Movement aborted due to#> : ').Append(_signalInfo.SymbolPath).As().AsError().Pin();
    _toHomePos := FALSE;
    IF (__ISVALIDREF(THIS^.inoToHomePos)) THEN
        THIS^.inoToHomePos := FALSE;
    END_IF;

    _moveHomeDefault.Abort();
END_IF
END_METHOD

(*~
    <docu>
        <summary>
            Aborts the movement to work position when the condition is 'true'.
        </summary>
        <remarks>
                <note type="warning">
                    The call of this method will be effective only when called AFTER the initialization of the instance of given TcoCylinder.
                </note>
        </remarks>
    </docu>
~*)
METHOD AbortMoveWork : BOOL
VAR_IN_OUT
    (*~
        <docu>
            <summary>
                Condition to abort the movement of the cylinder.
            </summary>
        </docu>
    ~*)
    inoDisableCondition : BOOL;
END_VAR
VAR
    _signalInfo : TcoSignalInfo;
END_VAR
IF (_toWorkPos OR _moveWorkDefault.Busy) AND inoDisableCondition THEN
    _signalInfo.GetSignalInfo(SIZEOF(inoDisableCondition), ADR(inoDisableCondition));
    Messenger.Build().Append('<#Movement aborted due to#> : ').Append(_signalInfo.SymbolPath).As().AsError().Pin();
    _toWorkPos := FALSE;
    IF (__ISVALIDREF(THIS^.inoToWorkPos)) THEN
        THIS^.inoToWorkPos := FALSE;
    END_IF;

    _moveWorkDefault.Abort();
END_IF
END_METHOD

(*~
    <docu>
        <summary>
            Gets the configuration of the cylinder.
        </summary>
    </docu>
~*)
PROPERTY Config : REFERENCE TO TcoCylinderConfig
GET
Config REF= _config;
END_GET
END_PROPERTY

(*~
    <docu>
        <summary>
            Gets the `MoveHomeTask` task that controls the moving of the cyclinder in home position.
        </summary>
    </docu>
~*)
PROPERTY MoveHomeTask : TcoCore.ITcoTask
GET
MoveHomeTask := _moveHomeDefault;
END_GET
END_PROPERTY

(*~
    <docu>
        <summary>
            Gets the `MoveWorkTask` task that controls the moving of the cyclinder into work position.
        </summary>
    </docu>
~*)
PROPERTY MoveWorkTask : TcoCore.ITcoTask
GET
MoveWorkTask := _moveWorkDefault;
END_GET
END_PROPERTY

(*~
    <docu>
        <summary>
            Refill cylinder after booth outputs are off .
        </summary>
        <remarks>
                <note type="warning">
                    The call of this method will be effective only when called AFTER the initialization of the instance of given TcoCylinder and methods like AbortMoveHone,SuspendMoveHom...
                </note>
        </remarks>
    </docu>
~*)
METHOD Refill : BOOL
VAR_INPUT
    (*~
    <docu>
        <summary>
            Time of refill cylinder after aborting or suspending
        </summary>
    </docu>
    ~*)
    inRefillTime : TIME;
END_VAR

_refillTimer(In := inoToHomePos XOR inoToWorkPos, Pt := T#49D);

_config.TimeToRefill := inRefillTime;

IF _refillTimer.ET > T#0MS
       AND _refillTimer.ET < _config.TimeToRefill
       AND _config.TimeToRefill <> T#0S THEN
    _toHomePos := TRUE;
    _toWorkPos := TRUE;
END_IF;

SUPER^
(
    inoAtHomePos1   := inoAtHomePos1
    , inoAtHomePos2 := inoAtHomePos2
    , inoAtWorkPos1 := inoAtWorkPos1
    , inoAtWorkPos2 := inoAtWorkPos2
    , inoToHomePos  := inoToHomePos
    , inoToWorkPos  := inoToWorkPos
);
END_METHOD

PROPERTY StatusCom : REFERENCE TO TcoCylinderStatus
GET
StatusCom REF= _status;
END_GET
END_PROPERTY

(*~
    <docu>
        <summary>
            Gets the `StopTask` task that controls the stopping of the cyclinder.
        </summary>
    </docu>
~*)
PROPERTY StopTask : TcoCore.ITcoTask
GET
StopTask := _stopDefault;
END_GET
END_PROPERTY

(*~
    <docu>
        <summary>
            Suspend the movement to home position when the condition is 'true'. Task is still busy
        </summary>
        <remarks>
                <note type="warning">
                    The call of this method will be effective only when called AFTER the initialization of the instance of given TcoCylinder.
                </note>
        </remarks>
    </docu>
~*)
METHOD SuspendMoveHome : BOOL
VAR_IN_OUT
    (*~
    <docu>
        <summary>
            Condition to abort the movement of the cylinder.
        </summary>
    </docu>
    ~*)
    inoDisableCondition : BOOL;
END_VAR
VAR
    _signalInfo : TcoSignalInfo;
END_VAR
IF (_toHomePos OR _moveHomeDefault.Busy) AND inoDisableCondition THEN
    _signalInfo.GetSignalInfo(SIZEOF(inoDisableCondition), ADR(inoDisableCondition));
    Messenger.Warning(CONCAT('<#Movement suspended due to#> : ', _signalInfo.SymbolPath));
    _toHomePos := FALSE;
    IF (__ISVALIDREF(THIS^.inoToHomePos)) THEN
        THIS^.inoToHomePos := FALSE;
    END_IF;

END_IF
END_METHOD

METHOD SuspendMoveHomeExpression : BOOL
VAR_INPUT
    inDisableCondition : BOOL;
    inMessage          : STRING;
END_VAR
IF (_toHomePos OR _moveHomeDefault.Busy) AND inDisableCondition THEN
    Messenger.Warning(CONCAT('<#Movement suspended due to#> : ', inMessage));
    _toHomePos := FALSE;
    IF (__ISVALIDREF(THIS^.inoToHomePos)) THEN
        THIS^.inoToHomePos := FALSE;
    END_IF;

END_IF;
END_METHOD

(*~
    <docu>
        <summary>
            Suspend the movement to home position when the condition is NOT 'true'. Task is still busy
        </summary>
        <remarks>
                <note type="warning">
                    The call of this method will be effective only when called AFTER the initialization of the instance of given TcoCylinder.
                </note>
        </remarks>
    </docu>
~*)
METHOD SuspendMoveHomeInverted : BOOL
VAR_IN_OUT
    (*~
    <docu>
        <summary>
            Condition to abort the movement of the cylinder.
        </summary>
    </docu>
    ~*)
    inoDisableCondition : BOOL;
END_VAR
VAR
    _signalInfo : TcoSignalInfo;
END_VAR
IF (_toHomePos OR _moveHomeDefault.Busy) AND NOT inoDisableCondition THEN
    _signalInfo.GetSignalInfo(SIZEOF(inoDisableCondition), ADR(inoDisableCondition));
    Messenger.Warning(CONCAT('<#Movement suspended due to NOT#> : ', _signalInfo.SymbolPath));
    _toHomePos := FALSE;
    IF (__ISVALIDREF(THIS^.inoToHomePos)) THEN
        THIS^.inoToHomePos := FALSE;
    END_IF;

END_IF
END_METHOD

(*~
    <docu>
        <summary>
            Suspend the movement to work position when the condition is 'true'. Task is still bussy
        </summary>
        <remarks>
                <note type="warning">
                    The call of this method will be effective only when called AFTER the initialization of the instance of given TcoCylinder.
                </note>
        </remarks>
    </docu>
~*)
METHOD SuspendMoveWork : BOOL
VAR_IN_OUT
    (*~
        <docu>
            <summary>
                Condition to abort the movement of the cylinder.
            </summary>
        </docu>
    ~*)
    inoDisableCondition : BOOL;
END_VAR
VAR
    _signalInfo : TcoSignalInfo;
END_VAR
IF (_toWorkPos OR _moveWorkDefault.Busy) AND inoDisableCondition THEN
    _signalInfo.GetSignalInfo(SIZEOF(inoDisableCondition), ADR(inoDisableCondition));
    Messenger.Warning(CONCAT('<#Movement suspended due to#> : ', _signalInfo.SymbolPath));
    _toWorkPos := FALSE;
    IF (__ISVALIDREF(THIS^.inoToWorkPos)) THEN
        THIS^.inoToWorkPos := FALSE;
    END_IF;

END_IF
END_METHOD

METHOD SuspendMoveWorkExpression : BOOL
VAR_INPUT
    inDisableCondition : BOOL;
    inMessage          : STRING;
END_VAR
IF (_toWorkPos OR _moveWorkDefault.Busy) AND inDisableCondition THEN
    Messenger.Warning(CONCAT('<#Movement suspended due to#> : ', inMessage));
    _toWorkPos := FALSE;
    IF (__ISVALIDREF(THIS^.inoToWorkPos)) THEN
        THIS^.inoToWorkPos := FALSE;
    END_IF;

END_IF
END_METHOD

(*~
    <docu>
        <summary>
            Suspend the movement to work position when the condition is NOT 'true'. Task is still bussy
        </summary>
        <remarks>
                <note type="warning">
                    The call of this method will be effective only when called AFTER the initialization of the instance of given TcoCylinder.
                </note>
        </remarks>
    </docu>
~*)
METHOD SuspendMoveWorkInverted : BOOL
VAR_IN_OUT
    (*~
        <docu>
            <summary>
                Condition to abort the movement of the cylinder.
            </summary>
        </docu>
    ~*)
    inoDisableCondition : BOOL;
END_VAR
VAR
    _signalInfo : TcoSignalInfo;
END_VAR
IF (_toWorkPos OR _moveWorkDefault.Busy) AND NOT inoDisableCondition THEN
    _signalInfo.GetSignalInfo(SIZEOF(inoDisableCondition), ADR(inoDisableCondition));
    Messenger.Warning(CONCAT('<#Movement suspended due to NOT#> : ', _signalInfo.SymbolPath));
    _toWorkPos := FALSE;
    IF (__ISVALIDREF(THIS^.inoToWorkPos)) THEN
        THIS^.inoToWorkPos := FALSE;
    END_IF;

END_IF
END_METHOD

END_FUNCTION_BLOCK

// ---- POUs/Cylinders/Zylinder/CylCustom.TcPOU
{attribute addProperty _moveHomeDefaultName "Home"} // Name/label of the move home task on HMI
{attribute addProperty _moveWorkDefaultName "Work"} // Name/label of the move work task on HMI
{attribute addProperty _stopDefaultName "Stop"}
FUNCTION_BLOCK CylCustom EXTENDS TcoPneumatics.TcoCylinderBase IMPLEMENTS iSuperActuator
VAR
    {attribute addProperty Name "|[[1]Attribute_moveWorkDefaultName]|"}
    _moveWorkDefault : CylCustomMoveTask(THIS^);
    {attribute addProperty Name "|[[1]Attribute_moveHomeDefaultName]|"}
    _moveHomeDefault : CylCustomMoveTask(THIS^);
    {attribute addProperty Name "|[[1]Attribute_stopDefaultName]|"}
    _stopDefault : TcoCore.TcoTask(THIS^);
    _faultTask   : TcoCore.TcoTask(THIS^);
END_VAR
VAR
    _config : TcoCylinderConfig;
    _status : TcoCylinderStatus;
    //~
    _watchDog : Tc2_Standard.TON;
    //~
    _watchDogTime              : TIME := T#3S;
    checkTimeBothSensorsActive : TIME := t#200ms;
END_VAR

SUPER^
(
    inoAtHomePos   := inoAtHomePos
    , inoAtWorkPos := inoAtWorkPos
    , inoToHomePos := inoToHomePos
    , inoToWorkPos := inoToWorkPos
);

_watchDog(in := (_atHomePos AND _atWorkPos) OR (NOT _atHomePos AND NOT _atWorkPos), PT := _watchDogTime);

IF _watchDog.ET > checkTimeBothSensorsActive THEN
    IF (_atHomePos AND _atWorkPos) THEN
        Messenger.Error('<#Home and work position sensors are both active. Check the position of sensors!#>')
            .Pin();

        _faultTask.ThrowWhen(_atHomePos AND _atWorkPos);
    END_IF
END_IF

IF _watchdog.Q THEN
    IF NOT _atHomePos AND NOT _atWorkPos THEN
        Messenger.Error('<#No Sensor Active, Check the position of the sensors!#>').Pin();
        _faultTask.ThrowWhen(NOT _atHomePos AND NOT _atWorkPos);
    END_IF;
END_IF;

// Disables mutualy exclusive actions
_moveWorkDefault.Enabled := NOT _moveHomeDefault.Busy;

_moveHomeDefault
(
    PositionSensor           := _atHomePos AND NOT _atWorkPos
    , MoveToPositionSignal   := _toHomePos
    , InverseSignal          := _toWorkPos
    , MaxTimeToReachPosition := _config.TimeToReachHomePosition
    , PositionName           := '<#Home#>'
);

// Disables mutualy exclusive actions
_moveHomeDefault.Enabled := NOT _moveWorkDefault.Busy;

_moveWorkDefault
(
    PositionSensor           := _atWorkPos AND NOT _atHomePos
    , MoveToPositionSignal   := _toWorkPos
    , InverseSignal          := _toHomePos
    , MaxTimeToReachPosition := _config.TimeToReachWorkPosition
    , PositionName           := '<#Work#>'
);

IF (_stopDefault.Execute()) THEN
    _toHomePos := FALSE;
    _toWorkPos := FALSE;
    _moveHomeDefault.Abort();
    _moveWorkDefault.Abort();
    _stopDefault.Abort();
    _moveHomeDefault.Restore();
    _moveWorkDefault.Restore();
    _stopDefault.Restore();
    _faultTask.Restore();
    _stopDefault.DoneWhen(TRUE);
END_IF

// For further discussion about Status
IF (_moveHomeDefault.Busy) THEN
    _status.ActionDescription := 'Moving to home position';
ELSIF (_moveWorkDefault.Busy) THEN
    _status.ActionDescription := 'Moving to work position';
ELSIF (_stopDefault.Busy) THEN
    _status.ActionDescription := 'Stopping pressure';
ELSIF (_moveHomeDefault.Error) THEN
    _status.ActionDescription := 'Error';
ELSIF (_moveWorkDefault.Error) THEN
    _status.ActionDescription := 'Error';
ELSIF (_faultTask.Error) THEN
    _status.ActionDescription := 'Error';
ELSE
    _status.ActionDescription := 'Idle';
END_IF

SUPER^
(
    inoAtHomePos   := inoAtHomePos
    , inoAtWorkPos := inoAtWorkPos
    , inoToHomePos := inoToHomePos
    , inoToWorkPos := inoToWorkPos
);

(*~
    <docu>
        <summary>
            Aborts the movement to home position when the condition is 'true'.
        </summary>
        <remarks>
                <note type="warning">
                    The call of this method will be effective only when called AFTER the initialization of the instance of given TcoCylinder.
                </note>
        </remarks>
    </docu>
~*)
METHOD AbortMoveHome : BOOL
VAR_IN_OUT
    (*~
    <docu>
        <summary>
            Condition to abort the movement of the cylinder.
        </summary>
    </docu>
    ~*)
    inoDisableCondition : BOOL;
END_VAR
VAR
    _signalInfo : TcoSignalInfo;
END_VAR
IF (_toHomePos OR _moveHomeDefault.Busy) AND inoDisableCondition THEN
    _signalInfo.GetSignalInfo(SIZEOF(inoDisableCondition), ADR(inoDisableCondition));
    Messenger.Error(CONCAT('<#Movement aborted due to#> : ', _signalInfo.SymbolPath));
    _toHomePos := FALSE;
    IF (__ISVALIDREF(THIS^.inoToHomePos)) THEN
        THIS^.inoToHomePos := FALSE;
    END_IF;

    _moveHomeDefault.Abort();
END_IF
END_METHOD

(*~
    <docu>
        <summary>
            Aborts the movement to work position when the condition is 'true'.
        </summary>
        <remarks>
                <note type="warning">
                    The call of this method will be effective only when called AFTER the initialization of the instance of given TcoCylinder.
                </note>
        </remarks>
    </docu>
~*)
METHOD AbortMoveWork : BOOL
VAR_IN_OUT
    (*~
        <docu>
            <summary>
                Condition to abort the movement of the cylinder.
            </summary>
        </docu>
    ~*)
    inoDisableCondition : BOOL;
END_VAR
VAR
    _signalInfo : TcoSignalInfo;
END_VAR
IF (_toWorkPos OR _moveWorkDefault.Busy) AND inoDisableCondition THEN
    _signalInfo.GetSignalInfo(SIZEOF(inoDisableCondition), ADR(inoDisableCondition));
    Messenger.Error(CONCAT('<#Movement aborted due to#> : ', _signalInfo.SymbolPath));
    _toWorkPos := FALSE;
    IF (__ISVALIDREF(THIS^.inoToWorkPos)) THEN
        THIS^.inoToWorkPos := FALSE;
    END_IF;

    _moveWorkDefault.Abort();
END_IF
END_METHOD

(*~
    <docu>
        <summary>
            Gets the configuration of the cylinder.
        </summary>
    </docu>
~*)
PROPERTY Config : REFERENCE TO TcoCylinderConfig
GET
Config REF= _config;
END_GET
END_PROPERTY

METHOD ErrorHandling : BOOL
//Messenger.Info('ErrorHandlingMetho');
END_METHOD

PROPERTY FaultTask : TcoCore.ITcoTask
GET
FaultTask := _faultTask;
END_GET
END_PROPERTY

PROPERTY IsError : BOOL
GET
IsError := MoveHomeTask.Error or MoveWorkTask.Error or FaultTask.Error;
END_GET
END_PROPERTY

PROPERTY PUBLIC MoveHomeTask : TcoCore.ITcoTask
GET
MoveHomeTask := _moveHomeDefault;
END_GET
END_PROPERTY

PROPERTY PUBLIC MoveWorkTask : TcoCore.ITcoTask
GET
MoveWorkTask := _moveWorkDefault;
END_GET
END_PROPERTY

METHOD ResetError : BOOL
VAR_INPUT
END_VAR
Restore();
END_METHOD

(*~
    <docu>
        <summary>
            Restore all tasks of this instance into initial state.
        </summary>
    </docu>
~*)
METHOD Restore : ITcoRestorable
SUPER^.Restore();
_watchDog(in := FALSE);

IF (MoveHomeTask <> 0) THEN
    MoveHomeTask.Restore();
END_IF;

IF (MoveWorkTask <> 0) THEN
    MoveWorkTask.Restore();
END_IF;

IF (StopTask <> 0) THEN
    StopTask.Restore();
END_IF;

IF (FaultTask <> 0) THEN
    FaultTask.Restore();
END_IF
END_METHOD

PROPERTY Status : REFERENCE TO TcoCylinderStatus
GET
Status REF= _status;
END_GET
END_PROPERTY

(*~
    <docu>
        <summary>
            Gets the `StopTask` task that controls the stopping of the cyclinder.
        </summary>
    </docu>
~*)
PROPERTY StopTask : TcoCore.ITcoTask
GET
StopTask := _stopDefault;
END_GET
END_PROPERTY

END_FUNCTION_BLOCK

// ---- POUs/Cylinders/Zylinder/CylCustomMoveTask.TcPOU
FUNCTION_BLOCK CylCustomMoveTask EXTENDS TcoCore.TcoTask
VAR_INPUT
    PositionSensor         : BOOL;
    MaxTimeToReachPosition : TIME := T#10S;
    PositionName           : STRING(25);
END_VAR
VAR_IN_OUT
    MoveToPositionSignal : BOOL;
    InverseSignal        : BOOL;
END_VAR

VAR
    _stringBuilder : TcoCore.StringBuilder;
END_VAR

IF (THIS^.Execute()) THEN
    IF (THIS^.ElapsedTime > MaxTimeToReachPosition) THEN
        THIS^.Messenger
            .Error(_stringBuilder.Clear().Append(PositionName).Append(' Sensor not reached, TimeOut!').ToString())
            .Pin();

        THIS^.ThrowWhen(TRUE);
    END_IF;

    InverseSignal        := FALSE;
    MoveToPositionSignal := TRUE;
    THIS^.DoneWhen(PositionSensor);
END_IF

METHOD PUBLIC FB_init : BOOL
VAR_INPUT
    bInitRetains : BOOL; // if TRUE, the retain variables are initialized (warm start / cold start)
    bInCopyCode  : BOOL; // if TRUE, the instance afterwards gets moved into the copy code (online change)
    ParentObject : ITcoObject;
END_VAR
// This is not clear to me... I from time to time the consumer code does not see 'FB_init' of 'TcoObject', that's why overridden here with super call...
SUPER^.FB_init(bInitRetains, bInCopyCode, ParentObject);
END_METHOD

(*~
    <docu>
        <summary>
            Executes when task is aborted.
        </summary>
    </docu>
~*)
METHOD PROTECTED OnAbort
MoveToPositionSignal := FALSE;
END_METHOD

METHOD PROTECTED OnError
THIS^.OnAbort();
END_METHOD

END_FUNCTION_BLOCK

// ---- POUs/Turck Rfid Reader/Rfid/Wrapper/Rfid_FB_Compact_Wrapper.TcPOU
FUNCTION_BLOCK Rfid_FB_Compact_Wrapper IMPLEMENTS IRfidHeadWrapper
VAR
    //Instantiate the function block
    turckRfid : RFID_FB_U.FB_Compact;

    // Create mapping to the I/O data of the corresponding channel
    stCompactModeInputMap  AT %I* : RFID_FB_U.CompactInput_t;
    stCompactModeOutputMap AT %Q* : RFID_FB_U.CompactOutput_t;
    // The Rx & Tx data mapping shown below is for example purposes only.
    // The actual array size can be 8,16,32,64 or 128 depending on slot configuration of the TBEC-LL-4RFID-8DXP box in the IO tree
    abyRxDataMapCompactMode AT %I* : ARRAY[0..127] OF BYTE;
    abyTxDataMapCompactMode AT %Q* : ARRAY[0..127] OF BYTE;
END_VAR

METHOD Execute
VAR_INPUT
    xExecute       : BOOL;
    xAbort         : BOOL;
    udiTimeOut     : UDINT;
    eCommand       : RFID_FB_U.COMMAND;
    udiStartAdress : UDINT;
    uiDataLenght   : UINT;
    myWriteData    : ARRAY[0..127] OF BYTE;
END_VAR
VAR_OUTPUT
    myReadData          : ARRAY[0..127] OF BYTE;
    xDone               : BOOL;
    xBusy               : BOOL;
    xError              : BOOL;
    xAborted            : BOOL;
    eErrorID            : RFID_FB_U.ERROR;
    xTP                 : BOOL;
    xRWHeadNotCOnnected : BOOL;
    uiDataRxLength      : UINT;
END_VAR
turckRfid
(
    xExecute              := xExecute
    , xAbort              := xAbort
    , udiTimeOut          := udiTimeOut
    , xDone               => xDone
    , xBusy               => xBusy
    , xError              => xError
    , xAborted            => xAborted
    , eCommand            := eCommand
    , rStatusMapping      := stCompactModeInputMap
    , rControlMapping     := stCompactModeOutputMap
    , udiStartAddress     := udiStartAdress
    , uiDataLength        := uiDataLenght
    , eErrorID            => eErrorID
    , xTP                 => xTP
    , xRWHeadNotConnected => xRWHeadNotCOnnected
    , uiDataRxLength      => uiDataRxLength
    , pReadDataMapping    := abyRxDataMapCompactMode
    , pWriteDataMapping   := abyTxDataMapCompactMode
    , pDataTx             := myWriteData
    , pDataRx             := myReadData
);
END_METHOD

END_FUNCTION_BLOCK

// ---- Project Information/F_GetCompany.TcPOU
// This function has been automatically generated from the project information.
{attribute 'signature_flag' := '1073741824'}
{attribute 'TcGenerated'}
{attribute 'no-analysis'}
FUNCTION F_GetCompany : WSTRING
VAR_INPUT

END_VAR

F_GetCompany := "Gema";

END_FUNCTION

// ---- Project Information/F_GetTitle.TcPOU
// This function has been automatically generated from the project information.
{attribute 'signature_flag' := '1073741824'}
{attribute 'TcGenerated'}
{attribute 'no-analysis'}
FUNCTION F_GetTitle : WSTRING
VAR_INPUT

END_VAR

F_GetTitle := "StandardLibGema";

END_FUNCTION

// ---- Project Information/F_GetVersion.TcPOU
// This function has been automatically generated from the project information.
{attribute 'signature_flag' := '1073741824'}
{attribute 'TcGenerated'}
{attribute 'no-analysis'}
FUNCTION F_GetVersion : ST_LibVersion
VAR_INPUT

END_VAR

F_GetVersion.iMajor    := 0;
F_GetVersion.iMinor    := 0;
F_GetVersion.iBuild    := 83;
F_GetVersion.iRevision := 0;
F_GetVersion.sVersion  := '0.0.83';
F_GetVersion.nFlags    := 0;

END_FUNCTION
